% RSLogix 500 project Conevor Belt That sort Object according to weight.RSS, saved by version 8.30.00.16 %
PROJECT "UNTITLED"    % processor: Bul.1763 MicroLogix 1100 Series B %

PROGRAM FILES
  LAD 2   4 rungs

DATA FILES
  O0 OUTPUT  4 elements
  I1 INPUT  6 elements
  S2 STATUS  66 elements
  B3 BINARY  1 elements
  T4 TIMER  1 elements
  C5 COUNTER  1 elements
  R6 CONTROL  1 elements
  N7 INTEGER  1 elements
  F8 FLOAT  1 elements

LADDER 2
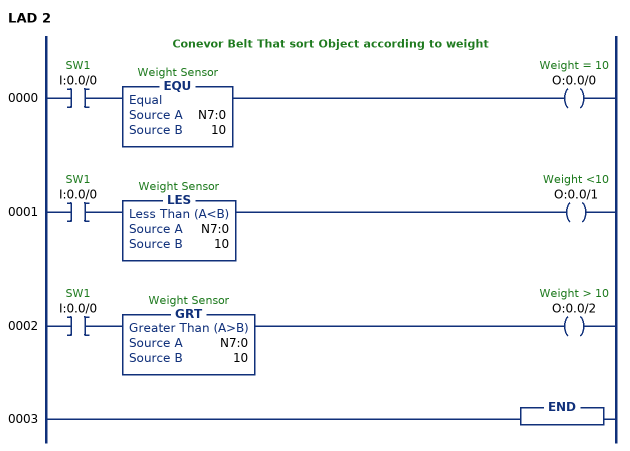
% Rung: 0 %
% TITLE: Conevor Belt That sort Object according to weight %
SOR XIC I:0.0/0 EQU N7:0 10 OTE O:0.0/0 EOR
%   I:0.0/0  "SW1" %
%   N7:0  "Weight Sensor" %
%   O:0.0/0  "Weight = 10" %
% Rung: 1 %
SOR XIC I:0.0/0 LES N7:0 10 OTE O:0.0/1 EOR
%   I:0.0/0  "SW1" %
%   N7:0  "Weight Sensor" %
%   O:0.0/1  "Weight <10" %
% Rung: 2 %
SOR XIC I:0.0/0 GRT N7:0 10 OTE O:0.0/2 EOR
%   I:0.0/0  "SW1" %
%   N7:0  "Weight Sensor" %
%   O:0.0/2  "Weight > 10" %
% Rung: 3 %
SOR END EOR

OTHER DOCUMENTED ADDRESSES
  I:0.0/1  "SW2"
  I:0.0/2  "SW2"
  I:0.0/3  "SW3"
  O:0.0/3  "Weight Not Equal to 10"

DATA TABLE (non-zero values as saved)
DATA N7
% N7:0 % 10
